PROGRAM MAIN
VAR
	stEventArray	: ARRAY[0..iNumEvents] OF ST_Event;
	
	
	bEstop			: BOOL :=TRUE;
	{attribute 'OPC.UA.DA' := '1'}
	bRun			: BOOL;
	{attribute 'TcAnalytics'}
	{attribute 'OPC.UA.DA' := '1'}
	rRealVal		: REAL;  //Process Value
	{attribute 'TcAnalytics'}
	bHeater			: BOOL;
	
	fbTON			: TON;
	{attribute 'TcAnalytics'}
	{attribute 'OPC.UA.DA' := '1'}
	bGoodCpk		: BOOL :=TRUE;
	lrRandom		: LREAL;
	iTmrPreset		: INT :=1000;
	iTmrET			: INT;
	fbDRAND			: DRAND;	
	rDutyCycle		: REAL :=50;

	sState			: STRING;
	sPrevState		: STRING;
	
	// date/time vars
    fbGetSystemTime  	: GETSYSTEMTIME;
    fileTimeUTC         : T_FILETIME;
    sDateTimeUTC        : STRING[32];

    fileTimeLocal       : T_FILETIME;
	systemTimeLocal		: TIMESTRUCT;
	sDateTimeLocal		: STRING[32];
	
	ulSysTime			: ULINT;

	myTime: DATE_AND_TIME;
	myTime2: TIME;
	myTime3: LTIME;
END_VAR

VAR CONSTANT
	iNumEvents: UINT := 99;
END_VAR

IF bEstop THEN
	bRun := FALSE;
	rRealVal := 50.0;
	bHeater := FALSE;
ELSE
	// run virtual machine
	IF bRun THEN
		fbDRAND(Seed:= iTmrET, Num=> lrRandom);
				
		IF bGoodCpk THEN
			rRealVal := 50 + 10 *(LREAL_TO_REAL(lrRandom)-0.5);
		ELSE
			rRealVal := rRealVal + 2 *(LREAL_TO_REAL(lrRandom)-0.5);
		END_IF
	END_IF	

	// Cycle heater based on duty cycle 	
	fbTON(IN:=NOT fbTON.q , PT:=INT_TO_TIME(iTmrPreset) , Q=> , ET=> );	
	iTmrET := TIME_TO_INT(fbTON.ET);
	
	IF iTmrET < iTmrPreset*rDutyCycle/100 THEN
		bHeater := TRUE;
	ELSE
		bHeater := FALSE;
	END_IF


END_IF

// Call EventLog action
aEventLog();

ACTION aEventLog:
// get timestamp
fbGetSystemTime(timeLoDW=>fileTimeUTC.dwLowDateTime, timeHiDW=>fileTimeUTC.dwHighDateTime);	// returns UTC time
sDateTimeUTC := SYSTEMTIME_TO_STRING(FILETIME_TO_SYSTEMTIME(fileTimeUTC));

// adjust for local timezone
//fileTimeLocal := F_TranslateFileTimeBias(in:= fileTime, bias:= WEST_EUROPE_TZI.bias + WEST_EUROPE_TZI.daylightBias, toUTC:= FALSE);
fileTimeLocal := F_TranslateFileTimeBias(in:= fileTimeUTC, bias:= 6*60, toUTC:= FALSE);
systemTimeLocal:=FILETIME_TO_SYSTEMTIME(fileTimeLocal);
sDateTimeLocal := SYSTEMTIME_TO_STRING(systemTimeLocal);

ulSysTime:=F_GetSystemTime();	// how to convert to string??

//Daymon playtime...
myTime := ULINT_TO_DT(ulSysTime);
myTime2 := ULINT_TO_TIME(ulSysTime);
myTime3 := ULINT_TO_LTIME(ulSysTime);


IF bEstop THEN
	sState := 'E-Stopped';
ELSE
	sState := 'Idle';	// default state if no Estop
	IF bRun THEN
		sState := 'Running';

		// ALARM - process out of spec - stop
		IF (rRealVal < 10) OR (rRealVal > 90) THEN
			bRun := FALSE;
			sState := 'Stopped - Out of Spec - Low!';
		END_IF
		IF (rRealVal > 90) THEN
			bRun := FALSE;
			sState := 'Stopped - Out of Spec - Hi!';
		END_IF

		// WARNING - process Cpk bad - but continue running
		IF sState = 'Running' THEN
			IF (rRealVal < 30) THEN
				sState := 'Running Low - Check Process!';
			END_IF
			IF (rRealVal > 70) THEN
				sState := 'Running High - Check Process!';
			END_IF
		END_IF
	END_IF
END_IF

(* Manage Event array... *)
IF sState <> sPrevState THEN	// if state change shift data down and add new event to top
	MEMMOVE(destAddr:= ADR(stEventArray[1]), srcAddr:= ADR(stEventArray[0]), n:= SIZEOF(stEventArray[0])*iNumEvents);

	(* current event values *)
	stEventArray[0].sDateTime := sDateTimeLocal;
	stEventArray[0].sEvent := sState;
	stEventArray[0].fProcVal := rRealVal;
	stEventArray[0].bHeaterState := bHeater;
END_IF
sPrevState := sState;
END_ACTION

END_PROGRAM

(* stored: Version 1.1.0.1, ProductVersion 3.1.4024.4
   POU MAIN: Id {f55654e8-ba50-4679-b5cf-b3d0778d83b0}, SpecialFunc None
   Action aEventLog: Id {44c1c4a0-45a8-4f4d-8a4c-b8182af57ec2} *)
